ABB RobotStudio station: Práctica4_inicio.rspag

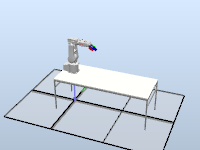
--- station ---
Station Práctica3_inicio (saved by RobotStudio 20.1.9056.2)
Controller Controlador2, task T_ROB1: task frame (RAPID world) sits at (0, 0, 670) mm in the station
Controller Controlador2
  mechanical unit ROB_1: IRB120_3_58__01, 6 joints, base frame (0, 0, 0) mm
Layout (positions relative to the parent item):
  - TVentosa [mechanism] at (364.35, 0, 1264) mm, rotated rx 180 ry 60 rz 180 deg
      TCP TVentosa at (0, 0, 51.19) mm
      links: Mi_herramienta
  - LogicGate [smart component, from Components\LogicGate.rslib]
      properties: Operator=NOT; Delay=0
  - LogicGate_2 [smart component, from Components\LogicGate.rslib]
      properties: Operator=AND; Delay=0
  - IRB120_3_58__01 [mechanism, from Robots\IRB120_3_58_G_01.rslib] at (0, 0, 670) mm; joint values [0, 0, 0, 0, 0.5236, 0] (rad or m)
  - table [part, from Libraries\e293a11e-ed86-4237-866f-a9bf8f4bd145table.rslib] at (-225, 300, 670) mm, rotated rx 0 ry 0 rz -90 deg
  - SimulationEvents [smart component, from Components\SimulationEvents.rslib]
Attachment: TVentosa is attached to IRB120_3_58__01 / Link6
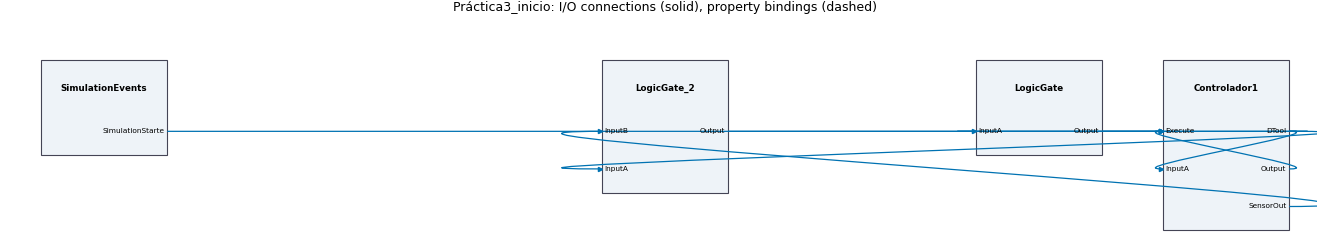
Station logic (signal -> signal, property => property):
  Controlador1.DTool -> Attacher.Execute
  Controlador1.DTool -> LogicGate_2.InputA
  LogicGate_2.Output -> Detacher.Execute
  Controlador1.DTool -> LogicGate.InputA
  LogicGate.Output -> Detacher.Execute
  CollisionSensor.SensorOut -> LogicGate_2.InputB
  Controlador1.DTool -> LogicGate_2.InputA
  LogicGate_2.Output -> Attacher.Execute
  SimulationEvents.SimulationStarted -> Source.Execute
Targets, tools, work objects and paths stored in the station and not in the controller backup, written as RAPID:
! task T_ROB1
MODULE CalibData
  PERS tooldata TVentosa:=[TRUE,[[0,0,51.19],[1,0,0,0]],[0.1,[0,0,1],[1,0,0,0],0,0,0]];
ENDMODULE


--- Backups/Controlador2/RAPID/TASK1/PROGMOD/Module1.mod ---
MODULE Module1
    !***********************************************************
    !
    ! Módulo:  Module1
    !
    ! Descripción:
    !   <Introduzca la descripción aquí>
    !
    ! Autor: Javier
    !
    ! Versión: 1.0
    !
    !***********************************************************


    !***********************************************************
    !
    ! Procedimiento Main
    !
    !   Este es el punto de entrada de su programa
    !
    !***********************************************************
    PROC main()
        !Añada aquí su código
    ENDPROC
ENDMODULE
